FUNCTION F_TimerEt2String : STRING
VAR_INPUT
	i_iTime				:TIME;
END_VAR
VAR
	iTimeInSec			:UDINT;
	iHours				:UDINT;
	iMinutes			:UDINT;
	iSeconds			:UDINT;
	sQuery				:STRING;
END_VAR

iTimeInSec:=TO_UDINT(i_iTIme)/1000;

iHours:=iTimeInSec/3600;
iMinutes:=(iTimeInSec/60)-(iHours*60);
iSeconds:=iTimeInSec - (iMinutes*60) - (iHours*3600);

IF iHours = 0 THEN
	sQuery:='00:';
ELSIF iHours > 0 AND iHours < 10 THEN
	sQuery:=CONCAT('0',TO_STRING(iHours));
	sQuery:=CONCAT(sQuery,':');
ELSE
	sQuery:=TO_STRING(iHours);
	sQuery:=CONCAT(sQuery,':');
END_IF

IF iMinutes = 0 THEN
	sQuery:=CONCAT(sQuery,'00:');
ELSIF iMinutes > 0 AND iMinutes < 10 THEN
	sQuery:=CONCAT(sQuery,'0');
	sQuery:=CONCAT(sQuery,TO_STRING(iMinutes));
	sQuery:=CONCAT(sQuery,':');
ELSE
	sQuery:=CONCAT(sQuery,TO_STRING(iMinutes));
	sQuery:=CONCAT(sQuery,':');
END_IF

IF iSeconds = 0 THEN
	sQuery:=CONCAT(sQuery,'00');
ELSIF iSeconds > 0 AND iSeconds < 10 THEN
	sQuery:=CONCAT(sQuery,'0');
	sQuery:=CONCAT(sQuery,TO_STRING(iSeconds));
ELSE
	sQuery:=CONCAT(sQuery,TO_STRING(iSeconds));
END_IF


F_TimerEt2String:=sQuery;

END_FUNCTION

(* stored: Version 1.1.0.1, ProductVersion 3.1.4024.12
   POU F_TimerEt2String: Id {e131ec3f-8ec0-45d6-ab55-e9400280978a}, SpecialFunc None *)
